PROGRAM MAIN
VAR
	iA: INT;
	iB: INT;
	iC: INT;
	
	fb_add1: FB_Add;
END_VAR

 fb_add1(iIn1:= iA, iIn2:= iB, iOut=> iC);

END_PROGRAM

(* stored: Version 1.1.0.1, ProductVersion 3.1.4024.12
   POU MAIN: Id {ca05b973-c3bc-4b90-a235-a0d338b80144}, SpecialFunc None *)
